SYSTEM EllipseFitting
  (* Version 1.0, 2020-07-24, LENOVO *)
  APPLICATION EllipseFittingApp
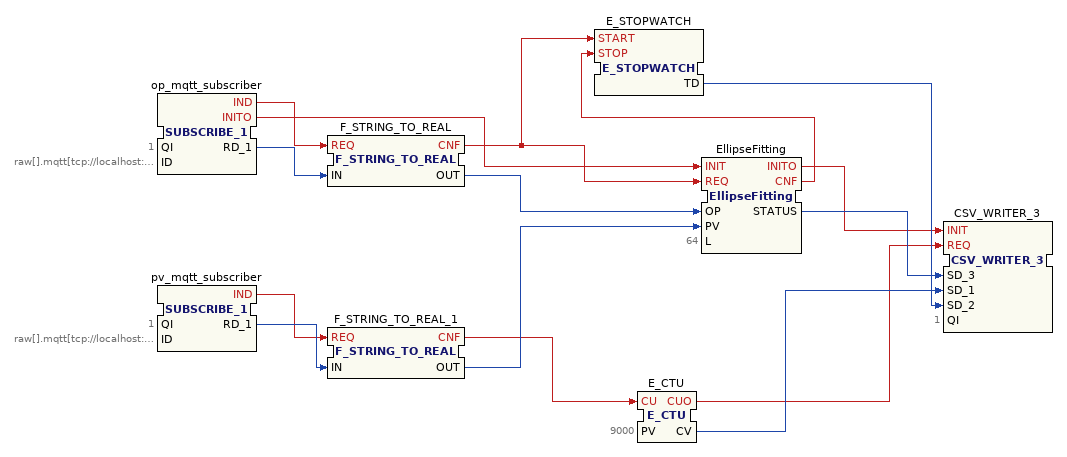
    FBS
      op_mqtt_subscriber : SUBSCRIBE_1(QI := 1, ID := raw[].mqtt[tcp://localhost:1883,forte,OP]);
      F_STRING_TO_REAL : F_STRING_TO_REAL;
      F_STRING_TO_REAL_1 : F_STRING_TO_REAL;
      pv_mqtt_subscriber : SUBSCRIBE_1(QI := 1, ID := raw[].mqtt[tcp://localhost:1883,forte,PV]);
      EllipseFitting : EllipseFitting(L := 64);
      E_CTU : E_CTU(PV := 9000);
      CSV_WRITER_3 : CSV_WRITER_3(QI := 1);
      E_STOPWATCH : E_STOPWATCH;
    END_FBS
    EVENT_CONNECTIONS
      op_mqtt_subscriber.IND TO F_STRING_TO_REAL.REQ;
      pv_mqtt_subscriber.IND TO F_STRING_TO_REAL_1.REQ;
      op_mqtt_subscriber.INITO TO EllipseFitting.INIT;
      F_STRING_TO_REAL_1.CNF TO E_CTU.CU;
      EllipseFitting.INITO TO CSV_WRITER_3.INIT;
      E_CTU.CUO TO CSV_WRITER_3.REQ;
      F_STRING_TO_REAL.CNF TO E_STOPWATCH.START;
      EllipseFitting.CNF TO E_STOPWATCH.STOP;
      F_STRING_TO_REAL.CNF TO EllipseFitting.REQ;
    END_CONNECTIONS
    DATA_CONNECTIONS
      pv_mqtt_subscriber.RD_1 TO F_STRING_TO_REAL_1.IN;
      op_mqtt_subscriber.RD_1 TO F_STRING_TO_REAL.IN;
      F_STRING_TO_REAL.OUT TO EllipseFitting.OP;
      F_STRING_TO_REAL_1.OUT TO EllipseFitting.PV;
      EllipseFitting.STATUS TO CSV_WRITER_3.SD_3;
      E_CTU.CV TO CSV_WRITER_3.SD_1;
      E_STOPWATCH.TD TO CSV_WRITER_3.SD_2;
    END_CONNECTIONS
  END_APPLICATION
  APPLICATION TestApp
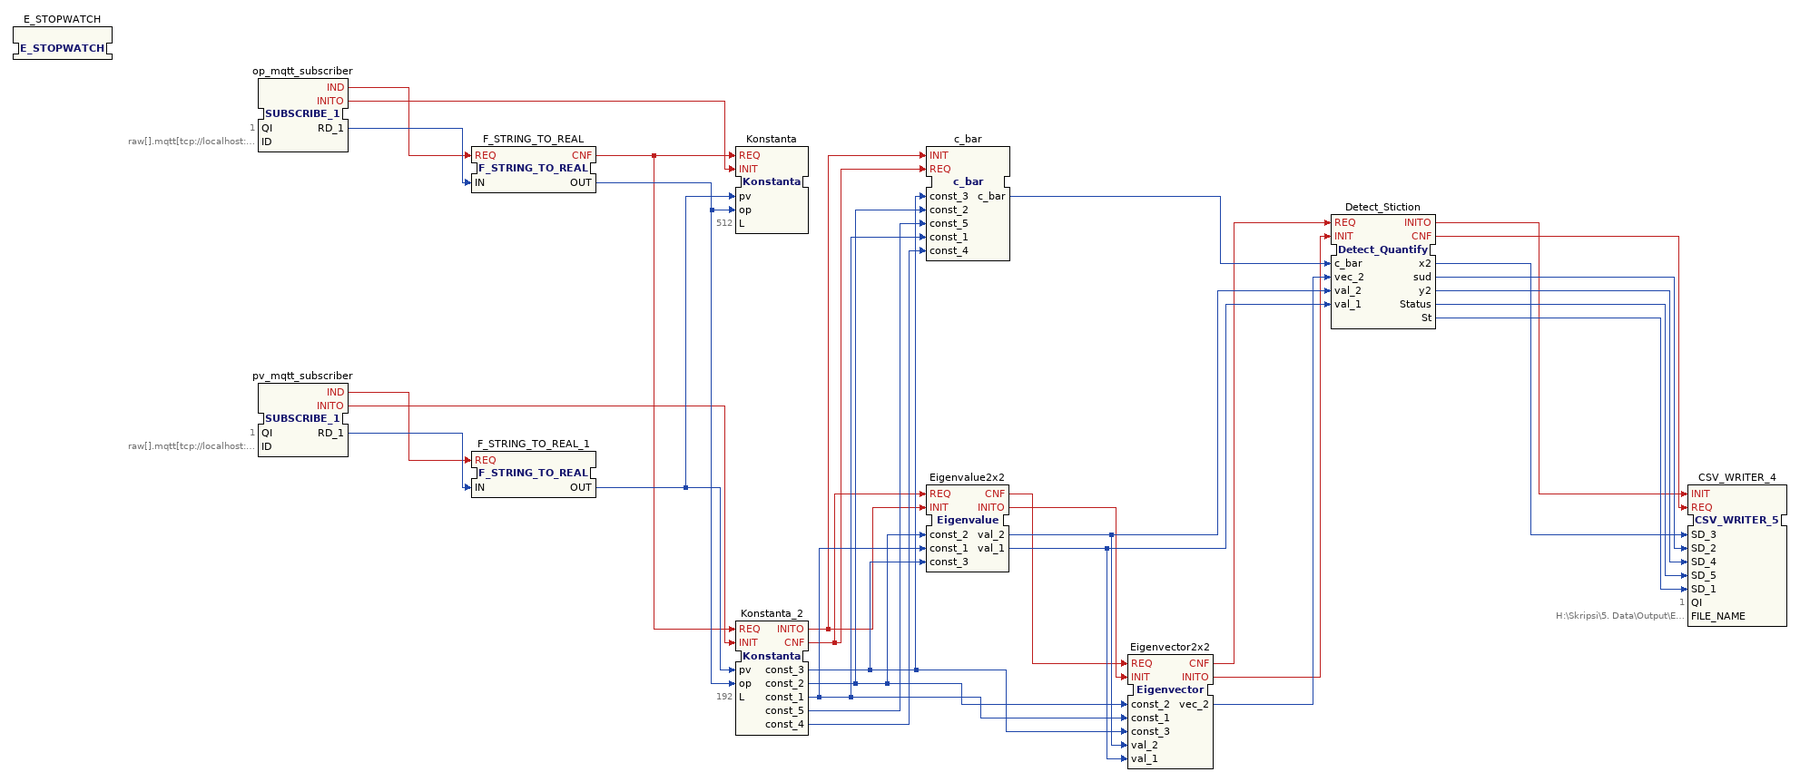
    FBS
      F_STRING_TO_REAL : F_STRING_TO_REAL;
      pv_mqtt_subscriber : SUBSCRIBE_1(QI := 1, ID := raw[].mqtt[tcp://localhost:1883,forte,PV]);
      op_mqtt_subscriber : SUBSCRIBE_1(QI := 1, ID := raw[].mqtt[tcp://localhost:1883,forte,OP]);
      Konstanta : Konstanta(L := 512);
      F_STRING_TO_REAL_1 : F_STRING_TO_REAL;
      c_bar : c_bar;
      Detect_Stiction : Detect_Quantify;
      Eigenvector2x2 : Eigenvector;
      Eigenvalue2x2 : Eigenvalue;
      CSV_WRITER_4 : CSV_WRITER_5(QI := 1, FILE_NAME := H:\Skripsi\5. Data\Output\EllipseFitting_192.csv);
      Konstanta_2 : Konstanta(L := 192);
      E_STOPWATCH : E_STOPWATCH;
    END_FBS
    EVENT_CONNECTIONS
      F_STRING_TO_REAL.CNF TO Konstanta.REQ;
      Konstanta_2.INITO TO c_bar.INIT;
      Konstanta_2.CNF TO Eigenvalue2x2.REQ;
      Konstanta_2.CNF TO c_bar.REQ;
      Detect_Stiction.INITO TO CSV_WRITER_4.INIT;
      F_STRING_TO_REAL.CNF TO Konstanta_2.REQ;
      op_mqtt_subscriber.IND TO F_STRING_TO_REAL.REQ;
      Detect_Stiction.CNF TO CSV_WRITER_4.REQ;
      Konstanta_2.INITO TO Eigenvalue2x2.INIT;
      Eigenvector2x2.CNF TO Detect_Stiction.REQ;
      Eigenvector2x2.INITO TO Detect_Stiction.INIT;
      op_mqtt_subscriber.INITO TO Konstanta.INIT;
      pv_mqtt_subscriber.IND TO F_STRING_TO_REAL_1.REQ;
      Eigenvalue2x2.CNF TO Eigenvector2x2.REQ;
      pv_mqtt_subscriber.INITO TO Konstanta_2.INIT;
      Eigenvalue2x2.INITO TO Eigenvector2x2.INIT;
    END_CONNECTIONS
    DATA_CONNECTIONS
      Detect_Stiction.x2 TO CSV_WRITER_4.SD_3;
      Detect_Stiction.sud TO CSV_WRITER_4.SD_2;
      F_STRING_TO_REAL_1.OUT TO Konstanta.pv;
      Konstanta_2.const_3 TO c_bar.const_3;
      F_STRING_TO_REAL_1.OUT TO Konstanta_2.pv;
      Konstanta_2.const_2 TO c_bar.const_2;
      Konstanta_2.const_2 TO Eigenvector2x2.const_2;
      c_bar.c_bar TO Detect_Stiction.c_bar;
      Detect_Stiction.y2 TO CSV_WRITER_4.SD_4;
      Konstanta_2.const_1 TO Eigenvector2x2.const_1;
      Konstanta_2.const_2 TO Eigenvalue2x2.const_2;
      op_mqtt_subscriber.RD_1 TO F_STRING_TO_REAL.IN;
      Konstanta_2.const_5 TO c_bar.const_5;
      Konstanta_2.const_3 TO Eigenvector2x2.const_3;
      Eigenvalue2x2.val_2 TO Eigenvector2x2.val_2;
      Konstanta_2.const_1 TO Eigenvalue2x2.const_1;
      Eigenvector2x2.vec_2 TO Detect_Stiction.vec_2;
      F_STRING_TO_REAL.OUT TO Konstanta_2.op;
      pv_mqtt_subscriber.RD_1 TO F_STRING_TO_REAL_1.IN;
      Eigenvalue2x2.val_1 TO Eigenvector2x2.val_1;
      Konstanta_2.const_1 TO c_bar.const_1;
      Eigenvalue2x2.val_2 TO Detect_Stiction.val_2;
      Detect_Stiction.Status TO CSV_WRITER_4.SD_5;
      Konstanta_2.const_3 TO Eigenvalue2x2.const_3;
      Konstanta_2.const_4 TO c_bar.const_4;
      Detect_Stiction.St TO CSV_WRITER_4.SD_1;
      Eigenvalue2x2.val_1 TO Detect_Stiction.val_1;
      F_STRING_TO_REAL.OUT TO Konstanta.op;
    END_CONNECTIONS
  END_APPLICATION
  DEVICE FORTE_PC : FORTE_PC(MGR_ID := "localhost:61499")
    {SET_ATTRIBUTE(Profile, HOLOBLOC)} (* device profile *)
    RESOURCE EMB_RES : EMB_RES
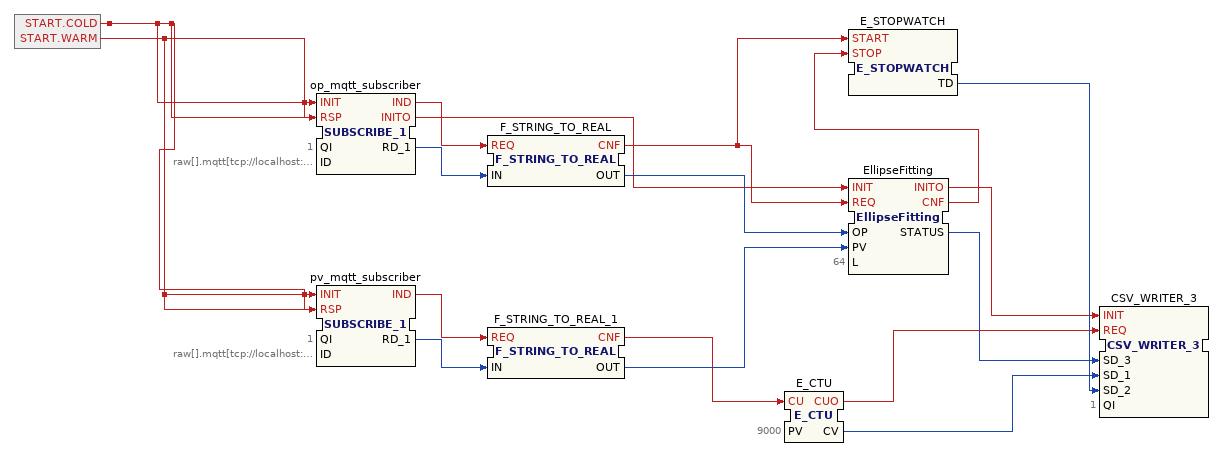
      FBS
        op_mqtt_subscriber : SUBSCRIBE_1(QI := 1, ID := raw[].mqtt[tcp://localhost:1883,forte,OP]);
        F_STRING_TO_REAL : F_STRING_TO_REAL;
        F_STRING_TO_REAL_1 : F_STRING_TO_REAL;
        pv_mqtt_subscriber : SUBSCRIBE_1(QI := 1, ID := raw[].mqtt[tcp://localhost:1883,forte,PV]);
        EllipseFitting : EllipseFitting(L := 64);
        E_CTU : E_CTU(PV := 9000);
        CSV_WRITER_3 : CSV_WRITER_3(QI := 1);
        E_STOPWATCH : E_STOPWATCH;
      END_FBS
      EVENT_CONNECTIONS
        op_mqtt_subscriber.IND TO F_STRING_TO_REAL.REQ;
        pv_mqtt_subscriber.IND TO F_STRING_TO_REAL_1.REQ;
        op_mqtt_subscriber.INITO TO EllipseFitting.INIT;
        F_STRING_TO_REAL_1.CNF TO E_CTU.CU;
        EllipseFitting.INITO TO CSV_WRITER_3.INIT;
        E_CTU.CUO TO CSV_WRITER_3.REQ;
        START.COLD TO op_mqtt_subscriber.INIT;
        START.WARM TO op_mqtt_subscriber.INIT;
        START.COLD TO op_mqtt_subscriber.RSP;
        START.WARM TO op_mqtt_subscriber.RSP;
        START.WARM TO pv_mqtt_subscriber.INIT;
        START.COLD TO pv_mqtt_subscriber.INIT;
        START.WARM TO pv_mqtt_subscriber.RSP;
        START.COLD TO pv_mqtt_subscriber.RSP;
        F_STRING_TO_REAL.CNF TO E_STOPWATCH.START;
        EllipseFitting.CNF TO E_STOPWATCH.STOP;
        F_STRING_TO_REAL.CNF TO EllipseFitting.REQ;
      END_CONNECTIONS
      DATA_CONNECTIONS
        op_mqtt_subscriber.RD_1 TO F_STRING_TO_REAL.IN;
        pv_mqtt_subscriber.RD_1 TO F_STRING_TO_REAL_1.IN;
        F_STRING_TO_REAL.OUT TO EllipseFitting.OP;
        F_STRING_TO_REAL_1.OUT TO EllipseFitting.PV;
        EllipseFitting.STATUS TO CSV_WRITER_3.SD_3;
        E_CTU.CV TO CSV_WRITER_3.SD_1;
        E_STOPWATCH.TD TO CSV_WRITER_3.SD_2;
      END_CONNECTIONS
    END_RESOURCE
  END_DEVICE
  MAPPINGS
    EllipseFittingApp.op_mqtt_subscriber ON FORTE_PC.EMB_RES.op_mqtt_subscriber;
    EllipseFittingApp.F_STRING_TO_REAL ON FORTE_PC.EMB_RES.F_STRING_TO_REAL;
    EllipseFittingApp.F_STRING_TO_REAL_1 ON FORTE_PC.EMB_RES.F_STRING_TO_REAL_1;
    EllipseFittingApp.pv_mqtt_subscriber ON FORTE_PC.EMB_RES.pv_mqtt_subscriber;
    EllipseFittingApp.EllipseFitting ON FORTE_PC.EMB_RES.EllipseFitting;
    EllipseFittingApp.E_CTU ON FORTE_PC.EMB_RES.E_CTU;
    EllipseFittingApp.CSV_WRITER_3 ON FORTE_PC.EMB_RES.CSV_WRITER_3;
    EllipseFittingApp.E_STOPWATCH ON FORTE_PC.EMB_RES.E_STOPWATCH;
  END_MAPPINGS
  SEGMENTS
    Ethernet : Ethernet;
  END_SEGMENTS
  LINKS
    FORTE_PC => Ethernet;
  END_LINKS
END_SYSTEM
